// TIA Portal project "Festo20230418" (V17)

(* hardware
DEVICE "S7-1200 station_1"  S7-1200 Station
   slot 0: "Rack_0"  S7-1200 Rack  Rack  V1.0
   slot 1: "PLC_1"  CPU 1214C AC/DC/Rly  6ES7 214-1BG40-0XB0  V4.5
   slot 3: "AQ 1x12BIT_1"  AQ1 signal board  6ES7 232-4HA30-0XB0  V1.0
DEVICE "S7-1200 station_2"  S7-1200 Station
   slot 0: "Rack_0"  S7-1200 Rack  Rack  V1.0
   slot 1: "PLC_2"  CPU 1215C AC/DC/Rly  6ES7 215-1BG40-0XB0  V4.5
   slot 3: "AQ 1x12BIT_1"  AQ1 signal board  6ES7 232-4HA30-0XB0  V1.0
*)

// ===== PLC "PLC_1"  CPU 1214C AC/DC/Rly =====

VAR_GLOBAL   // PLC tag table "Default tag table"
   "Clock_Byte" AT %MB0 : Byte;
   "Clock_10Hz" AT %M0.0 : Bool;
   "Clock_5Hz" AT %M0.1 : Bool;
   "Clock_2.5Hz" AT %M0.2 : Bool;
   "Clock_2Hz" AT %M0.3 : Bool;
   "Clock_1.25Hz" AT %M0.4 : Bool;
   "Clock_1Hz" AT %M0.5 : Bool;
   "Clock_0.625Hz" AT %M0.6 : Bool;
   "Clock_0.5Hz" AT %M0.7 : Bool;
   "System_Byte" AT %MB1 : Byte;
   "FirstScan" AT %M1.0 : Bool;
   "DiagStatusUpdate" AT %M1.1 : Bool;
   "AlwaysTRUE" AT %M1.2 : Bool;
   "AlwaysFALSE" AT %M1.3 : Bool;
   "FremVandret" AT %Q0.0 : Bool;
   "TilbageVandret" AT %Q0.1 : Bool;
   "NedLodret" AT %Q0.2 : Bool;
   "OpLodret" AT %Q0.3 : Bool;
   "Sug" AT %Q0.4 : Bool;
   "1S1 VandretTilbage" AT %I1.0 : Bool;
   "1S2 VandretFrem" AT %I1.1 : Bool;
   "2S1 Lodret Oppe" AT %I1.2 : Bool;
   "2S2 Lodret Nede" AT %I1.3 : Bool;
   "Tag_1" AT %IB0 : Byte;
   "Tag_2" AT %QB0 : Byte;
END_VAR

ORGANIZATION_BLOCK "Main"   // OB1, LAD, ProgramCycle
TITLE = "Main Program Sweep (Cycle)"
{ S7_Optimized_Access := 'TRUE' }
VERSION : 0.1
   VAR_INPUT
      Initial_Call : Bool;   // Initial call of this OB
      Remanence : Bool;   // =True, if remanent data are available
   END_VAR
BEGIN

REGION Network 2 (SCL)
   "Tag_2" := "Tag_1";
END_REGION
END_ORGANIZATION_BLOCK

// ===== PLC "PLC_2"  CPU 1215C AC/DC/Rly =====

VAR_GLOBAL   // PLC tag table "Default tag table"
   "System_Byte" AT %MB1 : Byte;
   "FirstScan" AT %M1.0 : Bool;
   "DiagStatusUpdate" AT %M1.1 : Bool;
   "AlwaysTRUE" AT %M1.2 : Bool;
   "AlwaysFALSE" AT %M1.3 : Bool;
   "Clock_Byte" AT %MB0 : Byte;
   "Clock_10Hz" AT %M0.0 : Bool;
   "Clock_5Hz" AT %M0.1 : Bool;
   "Clock_2.5Hz" AT %M0.2 : Bool;
   "Clock_2Hz" AT %M0.3 : Bool;
   "Clock_1.25Hz" AT %M0.4 : Bool;
   "Clock_1Hz" AT %M0.5 : Bool;
   "Clock_0.625Hz" AT %M0.6 : Bool;
   "Clock_0.5Hz" AT %M0.7 : Bool;
END_VAR

VAR_GLOBAL   // PLC tag table "IO_list"
   "Input_0" AT %I0.0 : Bool;
   "Input_1" AT %I0.1 : Bool;
   "Input_2" AT %I0.2 : Bool;
   "Input_3" AT %I0.3 : Bool;
   "Input_4" AT %I0.4 : Bool;
   "Input_5" AT %I0.5 : Bool;
   "Input_6" AT %I0.6 : Bool;
   "Input_7" AT %I0.7 : Bool;
   "Input_8" AT %I1.0 : Bool;
   "Input_9" AT %I1.1 : Bool;
   "Input_10" AT %I1.2 : Bool;
   "Input_11" AT %I1.3 : Bool;
   "Input_12" AT %I1.4 : Bool;
   "Input_13" AT %I1.5 : Bool;
   "Output_0" AT %Q0.0 : Bool;
   "Output_1" AT %Q0.1 : Bool;
   "Output_2" AT %Q0.2 : Bool;
   "Output_3" AT %Q0.3 : Bool;
   "Output_4" AT %Q0.4 : Bool;
   "Output_5" AT %Q0.5 : Bool;
   "Output_6" AT %Q0.6 : Bool;
   "Output_7" AT %Q0.7 : Bool;
   "Output_8" AT %Q1.0 : Bool;
   "Output_9" AT %Q1.1 : Bool;
   "AInput_0" AT %IW64 : Int;   // Voltage 0..10V
   "AInput_1" AT %IW66 : Int;   // Voltage 0..10V
   "AOutput_0" AT %QW64 : Int;   // Current 0..20mA
   "AOutput_1" AT %QW66 : Int;   // Current 0..20mA
   "AOutput_2" AT %QW80 : Int;   // Voltage 0..10V
END_VAR

DATA_BLOCK "DB_GlobalData"   // DB1
{ S7_Optimized_Access := 'TRUE' }
VERSION : 0.1
BEGIN
END_DATA_BLOCK

// folder: Unit

DATA_BLOCK "FB_Unit_EDUKIT_PA_Control_DB"   // DB2
{ S7_Optimized_Access := 'TRUE' }
VERSION : 0.1
// stored: InstanceOfName FB_Unit_EDUKIT_PA_Control
"FB_Unit_EDUKIT_PA_Control"
BEGIN
END_DATA_BLOCK

// folder: (top level)

ORGANIZATION_BLOCK "Main"   // OB1, LAD, ProgramCycle
TITLE = "Main Program Sweep (Cycle)"
{ S7_Optimized_Access := 'TRUE' }
VERSION : 0.1
   VAR_INPUT
      Initial_Call : Bool;   // Initial call of this OB
      Remanence : Bool;   // =True, if remanent data are available
   END_VAR
BEGIN
END_ORGANIZATION_BLOCK

// folder: Unit

FUNCTION_BLOCK "FB_Unit_EDUKIT_PA_Control"   // FB1, LAD
{ S7_Optimized_Access := 'TRUE' }
VERSION : 0.1
   VAR_INPUT
      Ainput_0 : Int;
      Ainput_1 : Int;
      Ainput_2 : Int;
   END_VAR
   VAR_OUTPUT
      output_startMotor : Bool;
      "output_motorPower [int]" : Int;
      output_valve : Bool;
   END_VAR
   VAR
      startMotor : Bool := true;
      "motorPower [%]" : Real := 85.0;
      valve : Bool;
      "Flow [l/h]" : Real;
      "pressure [mbar]" : Real;
      "pressure [psi]" : Real;
      "level [l]" : Real;
      "step" : Array[0..20] of Bool;
      PID_compact : PID_Compact;
   END_VAR
BEGIN

REGION Network 1
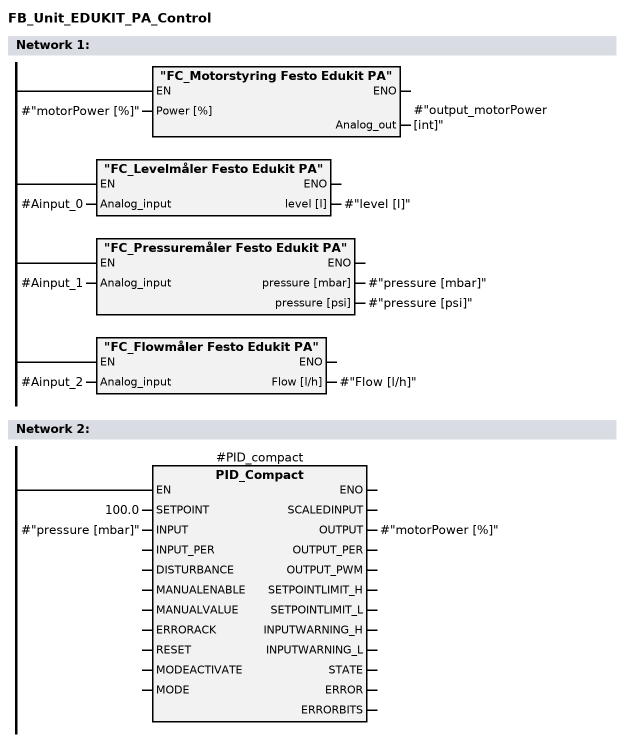
   RUNG wire#powerrail
      "FC_Motorstyring Festo Edukit PA"("Power [%]" := #"motorPower [%]", Analog_out => #"output_motorPower [int]")
   END_RUNG
   RUNG wire#powerrail
      "FC_Levelmåler Festo Edukit PA"(Analog_input := #Ainput_0, "level [l]" => #"level [l]")
   END_RUNG
   RUNG wire#powerrail
      "FC_Pressuremåler Festo Edukit PA"(Analog_input := #Ainput_1, "pressure [mbar]" => #"pressure [mbar]", "pressure [psi]" => #"pressure [psi]")
   END_RUNG
   RUNG wire#powerrail
      "FC_Flowmåler Festo Edukit PA"(Analog_input := #Ainput_2, "Flow [l/h]" => #"Flow [l/h]")
   END_RUNG
   // the same network as SCL:
   "FC_Motorstyring Festo Edukit PA"("Power [%]" := #"motorPower [%]", Analog_out => #"output_motorPower [int]");
   "FC_Levelmåler Festo Edukit PA"(Analog_input := #Ainput_0, "level [l]" => #"level [l]");
   "FC_Pressuremåler Festo Edukit PA"(Analog_input := #Ainput_1,
                           "pressure [mbar]" => #"pressure [mbar]",
                           "pressure [psi]" => #"pressure [psi]");
   "FC_Flowmåler Festo Edukit PA"(Analog_input := #Ainput_2, "Flow [l/h]" => #"Flow [l/h]");
END_REGION

REGION Network 2
   #PID_compact(Setpoint := 100.0, Input := #"pressure [mbar]", Output => #"motorPower [%]");   // PID_Compact
END_REGION

REGION Network 3 (SCL): Output_control
   IF #"output_motorPower [int]" > 30.0 THEN
       #output_startMotor := 1;
   ELSE
       #output_startMotor := 0;
   END_IF;

   #output_valve := 1;
END_REGION
END_FUNCTION_BLOCK

// folder: Unit/Control Modules

FUNCTION "FC_Motorstyring Festo Edukit PA" : Void   // FC1, SCL
{ S7_Optimized_Access := 'TRUE' }
VERSION : 0.1
   VAR_INPUT
      "Power [%]" : Real;   // Power 0.0..100.0%
   END_VAR
   VAR_OUTPUT
      Analog_out : Int;   // Analog output 0..27648
   END_VAR
   VAR_TEMP
      normPower : Real;   // Norm value 0.0..1.0
   END_VAR
   VAR CONSTANT
      minNorm_real : Real := 0.0;
      maxNorm_real : Real := 100.0;
      minScale_int : Int := 0;
      maxScale_int : Int := 27648;
   END_VAR
BEGIN
   (*
   norm and scale for motor controller on EDUKIT PA
   0.0..100.0%
   *)


   #Analog_out := SCALE_X_INT(
                              MIN := #minScale_int,
                              VALUE :=NORM_X_REAL(
                                                   MIN := #minNorm_real,
                                                   VALUE := #"Power [%]",
                                                   MAX := #maxNorm_real),
                              MAX := #maxScale_int);
END_FUNCTION

FUNCTION "FC_Flowmåler Festo Edukit PA" : Void   // FC2, SCL
{ S7_Optimized_Access := 'TRUE' }
VERSION : 0.1
   VAR_INPUT
      Analog_input : Int;   // Analog output 0..27648
   END_VAR
   VAR_OUTPUT
      "Flow [l/h]" : Real;   // Flow l/h
   END_VAR
   VAR_TEMP
      temp : Real;
   END_VAR
   VAR CONSTANT
      minNorm_int : Int := 0;
      maxNorm_int : Int := 27648;
      minScale_real : Real := 0.0;
      maxScale_real : Real := 100.0;
   END_VAR
BEGIN
   (*
   norm and scale for flow sensor on EDUKIT PA
   0..10V 0..400 mbar
   *)

   #temp:=NORM_X_REAL(MIN := #minNorm_int, VALUE := #Analog_input, MAX := #maxNorm_int);
   #"Flow [l/h]" := 463.9 * #temp - 7.8427;
   IF #"Flow [l/h]" < 0.0 THEN
       #"Flow [l/h]" := 0;
   END_IF;
   (*
   measurements
   norm[%] l/h
   0,275   120
   0,320   140
   0,361   160
   0,405   180

   y = 463,9x - 7,8427
   R² = 0,9997

   *)
END_FUNCTION

FUNCTION "FC_Pressuremåler Festo Edukit PA" : Void   // FC3, SCL
{ S7_Optimized_Access := 'TRUE' }
VERSION : 0.1
   VAR_INPUT
      Analog_input : Int;   // Analog output 0..27648
   END_VAR
   VAR_OUTPUT
      "pressure [mbar]" : Real;   // pressure bar 0..400mbar
      "pressure [psi]" : Real;   // pressure psi
   END_VAR
   VAR_TEMP
      temp : Real;
   END_VAR
   VAR CONSTANT
      minNorm_int : Int := 0;
      maxNorm_int : Int := 27648;
      minScale_real : Real := 0.0;
      maxScale_real : Real := 100.0;
   END_VAR
BEGIN
   (*
   norm and scale for pressure sensor on EDUKIT PA
   0..10V 0..400 mbar
   1 millibar = 0.0145037738 psi
   *)

   #temp:=NORM_X_REAL(MIN := #minNorm_int, VALUE := #Analog_input, MAX := #maxNorm_int);
   #"pressure [mbar]" := 400.0 * #temp;
   #"pressure [psi]" := #"pressure [mbar]" * 0.0145037738;
END_FUNCTION

FUNCTION "FC_Levelmåler Festo Edukit PA" : Void   // FC4, SCL
{ S7_Optimized_Access := 'TRUE' }
VERSION : 0.1
   VAR_INPUT
      Analog_input : Int;   // Analog output 0..27648
   END_VAR
   VAR_OUTPUT
      "level [l]" : Real;   // Flow l/h
   END_VAR
   VAR_TEMP
      temp : Real;
   END_VAR
   VAR CONSTANT
      minNorm_int : Int := 0;
      maxNorm_int : Int := 27648;
      minScale_real : Real := 0.0;
      maxScale_real : Real := 100.0;
   END_VAR
BEGIN
   (*
   norm and scale for level sensor on EDUKIT PA
   0..10V 0..2.7 liters
   *)

   #temp:=NORM_X_REAL(MIN := #minNorm_int, VALUE := #Analog_input, MAX := #maxNorm_int);
   #"level [l]" := 2.7 * #temp;
   IF #"level [l]" < 0.0 THEN
       #"level [l]" := 0;
   END_IF;
   (*
   measurements
   norm[%] l
   0,275   
   0,320   
   0,361   
   0,405   

   *)
END_FUNCTION